// TwinCAT 3 PLC project TwinCAT_OpenFramework_JSON
// Title: TwinCAT Open Framework JSON
// Company: Oleksandr Tiutyk FOP
// Author: Oleksandr Tiutyk
// ProjectVersion: 1.0.13.0
// Description: TwinCAT.OpenFramework сlasses that help in working with JSON
// ProgramVersion: 3.1.4026.28
// libraries:
//   Tc2_Utilities, * (Beckhoff Automation GmbH)
//   Tc3_JsonXml, * (Beckhoff Automation GmbH)
//   [TwinCAT Open Framework Core], * (Oleksandr Tiutyk FOP)
// project tree:
//   AutomaticSerializer/ AutomaticJsonSerializer.TcPOU, IJsonExtender.TcIO
//   Configuration/ JsonConfigurationReader.TcPOU, JsonConfigurationWriter.TcPOU
//   Internal/ CurrentNamespace.TcPOU, JsonDatatypes.TcPOU, NamespaceExtractor.TcPOU
//   Version/ Global_Version.TcGVL
// (motion and I/O tree: see PLC project twincat_openframework_core)
// real-time tasks:
//   TASK PlcTask: cycle T#10ms, priority 20, ADS port 350
//   TASK TestTask: cycle T#10ms, priority 1, ADS port 351
//   TASK RunnerTestTask: cycle T#10ms, priority 2, ADS port 354
//   TASK HowToTask: cycle T#10ms, priority 22, ADS port 353
// variable links:

// ---- Version/Global_Version.TcGVL
{attribute 'TcGenerated'}
{attribute 'no-analysis'}
{attribute 'linkalways'}
// This function has been automatically generated from the project information.
VAR_GLOBAL CONSTANT
	{attribute 'const_non_replaced'}
	stLibVersion_TwinCAT_Open_Framework_JSON : ST_LibVersion := (iMajor := 1, iMinor := 0, iBuild := 13, iRevision := 0, nFlags := 0, sVersion := '1.0.13.0');
END_VAR

// ---- AutomaticSerializer/IJsonExtender.TcIO
(*
SPDX-FileCopyrightText: © 2026 Oleksandr Tiutyk <trofimich@gmail.com>
SPDX-License-Identifier: MIT
License: https://opensource.org/license/mit
*)

(*!
<summary>Extends serialization by writing around the structure's JSON value.</summary>
<description>
AutomaticJsonSerializer calls these hooks synchronously on its own SAX writer. The writer belongs to the
serializer; callbacks do not acquire ownership. The combined hook output and structure value must form the
intended JSON document. The writer is borrowed only for the duration of each callback and must not be retained
or handed to another task. Hooks execute in the serializer's owner task. Do not call methods or access
properties of the active serializer, directly or indirectly; a nested conversion needs a separate serializer
and separate buffers. Stateful extenders must not be used concurrently by different tasks. Implementations
handle failures reported by the native methods they invoke. Callback exceptions propagate from Create methods
and are contained by TrySerialize methods; prior writes and external callback effects are not rolled back.
WriteSuffix is not a cleanup or finally callback.
</description>
*)
INTERFACE IJsonExtender

(*!
<summary>Writes the prefix before serialization of the structure value.</summary>
<description>
Called after successful ResetDocument, before AddJsonValueFromSymbol. Leave the writer ready to receive the
structure as a JSON value, for example after an enclosing container's key. A later failure does not guarantee a
WriteSuffix call or roll back callback effects.
</description>
<param name="jsonSaxWriter">Serializer-owned writer reset for the current conversion.</param>
*)
METHOD WritePrefix
VAR_IN_OUT CONSTANT
	jsonSaxWriter : Tc3_JsonXml.FB_JsonSaxWriter;	
END_VAR
END_METHOD

(*!
<summary>Writes the suffix after successful serialization of the structure value.</summary>
<description>
Called before copying the document to the caller's buffer. May finish a container opened by WritePrefix. It
is skipped if reset, the start hook or structure serialization fails, including terminal allocation failure
contained inside a hook. Later copy failure does not roll back its effects.
</description>
<param name="jsonSaxWriter">Serializer-owned writer containing the prefix and structure value.</param>
*)
METHOD WriteSuffix
VAR_IN_OUT CONSTANT
	jsonSaxWriter : Tc3_JsonXml.FB_JsonSaxWriter;	
END_VAR
END_METHOD

END_INTERFACE

// ---- AutomaticSerializer/AutomaticJsonSerializer.TcPOU
(*
SPDX-FileCopyrightText: © 2026 Oleksandr Tiutyk <trofimich@gmail.com>
SPDX-License-Identifier: MIT
License: https://opensource.org/license/mit
*)

(*!
<summary>Serializes live PLC structures to JSON and restores them from JSON.</summary>
<description>
Supports live PLC structures with native type information; dynamically created structures are not supported.
ByVarInfo methods require an explicit PVOID address; descriptor ByteAddress is ignored to preserve pointer width.
Application method calls and property access belong to one owner task per instance. Instances are not
thread-safe and do not support reentry: a callback must not call methods or access properties of the
serializer whose operation is still active, directly or indirectly. Use a separate instance and separate
buffers for another task or nested conversion. Ownership is a caller precondition, not a runtime check or
lock; Try does not make an ownership violation safe or guarantee its detection as FALSE. Keep source data
stable and destination storage exclusive for the entire call, including callbacks. Separate serializer
instances do not synchronize shared application data. Stateful extenders require their own ownership
discipline; sharing an extender must not introduce concurrent state access. Borrows input, output and optional
callbacks for each call. Throwing methods report invalid arguments and native failures through framework
exceptions. Try methods return FALSE directly for rejected arguments or reported native failures and contain
exceptions from native calls or callbacks; partial effects are not rolled back. Try methods use the shared
native conversion helpers, not overrides of the throwing methods or their protected helpers. JSON text uses
native UTF-8 encoding; capacity and copy sizes count bytes. Instances must not be copied by value. The caller
provides cyclic-task exception cleanup and RaiseIfAllocationFailed at the task boundary, outside Try and
recoverable handlers. Try methods do not clear terminal allocation state. Ownership examples and future
shared-service guidance: Guides/JsonAndEventLoggerOwnership.md in the repository.
</description>
*)

{attribute 'no_explicit_call' := 'Direct call is not allowed'}
FUNCTION_BLOCK AutomaticJsonSerializer EXTENDS TOF_Core.Object
VAR_STAT
	//! <summary>Class name shared by all instances of this function block.</summary>
	{attribute 'hide'} 
	_ClassName : STRING := __POUNAME();
END_VAR
VAR
	_JsonSaxWriter : Tc3_JsonXml.FB_JsonSaxWriter;
	_JsonDataTypeWriter : Tc3_JsonXml.FB_JsonReadWriteDatatype;
END_VAR

(*!
<summary>Provides the concrete serializer class name.</summary>
<description>Borrows read-only instance storage that remains valid for the instance lifetime.</description>
*)
{attribute 'monitoring' := 'call'}
PROPERTY ClassName : REFERENCE TO STRING
GET
ClassName REF= _ClassName;
END_GET
END_PROPERTY

(*!
<summary>Serializes a PLC structure into caller-owned JSON storage.</summary>
<description>
Uses native symbol lookup for the source type; dynamically created structures are not supported. Single-field
structures have native lookup limitations; use ByVarInfo to supply the type explicitly. Borrows
source, destination and optional extender for the call. The destination must be writable and have at least
JSON_DOCUMENT capacity. Invalid source arguments and reported native failures raise framework exceptions;
extender exceptions propagate. Output and callback effects are not rolled back on failure. Exception transport
and cleanup require the caller's cyclic-task boundary. CopyDocument returning zero or a nonzero HRESULT raises
an exception; jsonSize is not usable on failure.
</description>
<param name="sourceStructure">Live PLC structure with type information available to native symbol lookup.</param>
<param name="extender">
Optional callback invoked before and after writing the structure value; zero skips both calls.
</param>
<param name="targetJson">Writable output storage with at least 25000 bytes of text capacity plus the terminator.</param>
<param name="jsonSize">
Byte count reported by CopyDocument, including the terminator on a successful copy; use only after normal
completion.
</param>
*)
METHOD Serialize
VAR_INPUT
	sourceStructure : ANY;
	extender : IJsonExtender := 0;
END_VAR
VAR_IN_OUT
	targetJson : TOF_Core.JSON_DOCUMENT;
END_VAR
VAR_OUTPUT
	jsonSize : UDINT; 
END_VAR
InternalSerialize(
	sourceStructure := sourceStructure,
	extender := extender,
	targetJson := targetJson,
	jsonSize => jsonSize
);
END_METHOD

(*!
<summary>Serializes a PLC structure described by VAR_INFO into caller-owned JSON storage.</summary>
<description>
The descriptor type and byte-aligned size must match sourceStructureAddress. ByteAddress is ignored.
Dynamically created structures are not supported. Borrows source, destination and optional extender for the call. The
destination must be writable and have at least JSON_DOCUMENT capacity. Invalid source arguments and reported
native failures raise framework exceptions; extender exceptions propagate. Output and callback effects are not
rolled back on failure. Exception transport and cleanup require the caller's cyclic-task boundary.
CopyDocument returning zero or a nonzero HRESULT raises an exception; jsonSize is not usable on failure.
</description>
<param name="sourceStructureAddress">
Required address from ADR of the live source structure, borrowed for this call. Must match the descriptor.
Zero is rejected; no address is recovered from ByteAddress or ByteOffset.
</param>
<param name="sourceStructureVarInfo">
Descriptor whose TypeName and BitSize describe the source structure; ByteAddress is ignored.
</param>
<param name="extender">
Optional callback invoked before and after writing the structure value; zero skips both calls.
</param>
<param name="targetJson">Writable output storage with at least 25000 bytes of text capacity plus the terminator.</param>
<param name="jsonSize">
Byte count reported by CopyDocument, including the terminator on a successful copy; use only after normal
completion.
</param>
*)
METHOD SerializeByVarInfo
VAR_INPUT
	sourceStructureVarInfo : __SYSTEM.VAR_INFO;
	sourceStructureAddress : PVOID;
	extender : IJsonExtender := 0;
END_VAR
VAR_IN_OUT
	targetJson : TOF_Core.JSON_DOCUMENT;
END_VAR
VAR_OUTPUT
	jsonSize : UDINT; 
END_VAR
VAR
	formattedExceptionMessage : TOF_Core.ERROR_MESSAGE;

	
	errorCode : HRESULT;
END_VAR
IF sourceStructureAddress = TOF_Core.Memory.NULL_ADDRESS THEN
	TOF_Core.Exceptions.ThrowArgumentNotSpecified(
		sourceNamespaceName := NamespaceName,
		sourceClassName := ClassName,
		sourcePOUName := __POUNAME(),
		sourcePosition := __POSITION(),
		argumentName := 'sourceStructureAddress'
	);
END_IF

IF sourceStructureVarInfo.TypeClass <> __SYSTEM.TYPE_CLASS.TYPE_USERDEF THEN
	TOF_Core.Exceptions.ThrowArgumentTypeClassNotSupported(
		sourceNamespaceName := NamespaceName,
		sourceClassName := ClassName,
		sourcePOUName := __POUNAME(),
		sourcePosition := __POSITION(),
		argumentName := 'sourceStructureVarInfo',
		argumentType := sourceStructureVarInfo.TypeClass
	);
END_IF

// VAR_INFO sizes are in bits; the caller supplies a byte-aligned structure descriptor.
IF NOT writeStructureJson(
	structureTypeName := sourceStructureVarInfo.TypeName,
	structureAddress := sourceStructureAddress,
	structureSize := TO_UDINT(sourceStructureVarInfo.BitSize / 8),
	extender := extender,
	targetJson := targetJson,
	jsonSize => jsonSize,
	errorCode => errorCode,
	errorMessage => formattedExceptionMessage
)
THEN
	TOF_Core.Exceptions.ThrowStandard(
		sourceNamespaceName := NamespaceName,
		sourceClassName := ClassName,
		sourcePOUName := __POUNAME(),
		sourcePosition := __POSITION(),
		message := formattedExceptionMessage,
		errorCode := TO_UDINT(errorCode)
	);
END_IF
END_METHOD

{attribute 'monitoring' := 'call'}
(*!
<summary>Gets or sets the native writer's maximum number of fractional decimal places.</summary>
<description>
The native writer determines which DINT values it supports; this property does not clamp the value. The setter
requires a zero HRESULT from SetMaxDecimalPlaces. A nonzero HRESULT raises a framework exception because
assignment has no failure result. The native error code is retained in the exception. No rollback of the
native setting is guaranteed on failure; the getter reads the writer's current setting. The caller handles the
exception and provides cyclic-task exception cleanup and the terminal allocation-failure boundary.
</description>
*)
PROPERTY DecimalPlaces : DINT
GET
DecimalPlaces := _JsonSaxWriter.GetMaxDecimalPlaces();
END_GET
SET
VAR
	errorCode : HRESULT;
END_VAR
errorCode := _JsonSaxWriter.SetMaxDecimalPlaces(decimalPlaces := DecimalPlaces);

IF errorCode <> TOF_Core.SignedInt32.ZERO THEN
	TOF_Core.Exceptions.ThrowStandard(
		sourceNamespaceName := NamespaceName,
		sourceClassName := ClassName,
		sourcePOUName := __POUNAME(),
		sourcePosition := __POSITION(),
		message := "Can't set JSON writer decimal places",
		errorCode := TO_UDINT(errorCode)
	);
END_IF
END_SET
END_PROPERTY

(*!
<summary>Populates a PLC structure from JSON using the type supplied by VAR_INFO.</summary>
<description>
TypeName and byte-aligned BitSize must describe the live, writable structure at targetStructureAddress.
ByteAddress is ignored. Uses the supplied TypeName directly, avoiding ambiguous address-based type lookup
for single-field structures. The type
must be available to the native JSON converter; support for dynamically created structures is not implied.
Borrows the JSON and destination for this call. A zero address, an unsupported type class or a reported native
conversion failure raises a framework exception. Conversion requires both a TRUE SetSymbolFromJson result and
a zero HRESULT. Destination fields may already have changed on failure; writes are not rolled back. The caller
provides cyclic-task exception cleanup and the terminal allocation-failure boundary.
</description>
<param name="json">JSON text to read without modification.</param>
<param name="targetStructureAddress">
Required address from ADR of the live target structure, borrowed for this call. Must match the descriptor.
Zero is rejected; no address is recovered from ByteAddress or ByteOffset.
</param>
<param name="targetStructureVarInfo">
Consistent descriptor of the destination structure, including its explicit TypeName.
</param>
*)
METHOD DeserializeByVarInfo
VAR_IN_OUT CONSTANT
	json : TOF_Core.JSON_DOCUMENT;	
END_VAR
VAR_INPUT
	targetStructureVarInfo : __SYSTEM.VAR_INFO;
	targetStructureAddress : PVOID;
END_VAR
VAR
	
	errorCode : HRESULT;
END_VAR
IF targetStructureAddress = TOF_Core.Memory.NULL_ADDRESS THEN
	TOF_Core.Exceptions.ThrowArgumentNotSpecified(
		sourceNamespaceName := NamespaceName,
		sourceClassName := ClassName,
		sourcePOUName := __POUNAME(),
		sourcePosition := __POSITION(),
		argumentName := 'targetStructureAddress'
	);
END_IF

IF targetStructureVarInfo.TypeClass <> __SYSTEM.TYPE_CLASS.TYPE_USERDEF THEN
	TOF_Core.Exceptions.ThrowArgumentTypeClassNotSupported(
		sourceNamespaceName := NamespaceName,
		sourceClassName := ClassName,
		sourcePOUName := __POUNAME(),
		sourcePosition := __POSITION(),
		argumentName := 'targetStructureVarInfo',
		argumentType := targetStructureVarInfo.TypeClass
	);
END_IF

// VAR_INFO sizes are in bits; the caller supplies a byte-aligned structure descriptor.
IF NOT readStructureJson(
	json := json,
	structureTypeName := targetStructureVarInfo.TypeName,
	structureAddress := targetStructureAddress,
	structureSize := TO_UDINT(targetStructureVarInfo.BitSize / 8),
	errorCode => errorCode
)
THEN
	TOF_Core.Exceptions.ThrowStandard(
		sourceNamespaceName := NamespaceName,
		sourceClassName := ClassName,
		sourcePOUName := __POUNAME(),
		sourcePosition := __POSITION(),
		message := "Can't fill target structure by specified json document",
		errorCode := TO_UDINT(errorCode)
	);
END_IF
END_METHOD

(*!
<summary>Populates a PLC structure from JSON using native address-based type lookup.</summary>
<description>
Borrows the JSON and a live, writable structure for the call; dynamically created structures are not
supported. Native type lookup has limitations for single-field structures. Invalid arguments, reported lookup
failures, a FALSE SetSymbolFromJson result or a nonzero conversion HRESULT raise framework exceptions.
Destination fields may already have changed on failure; writes are not rolled back. The caller provides
cyclic-task exception cleanup and the terminal allocation-failure boundary.
</description>
<param name="json">JSON text to read without modification.</param>
<param name="targetStructure">
Live destination structure with type information available to native symbol lookup.
</param>
*)
METHOD Deserialize
VAR_IN_OUT CONSTANT
	json : TOF_Core.JSON_DOCUMENT;	
END_VAR
VAR_INPUT
	targetStructure : ANY;
END_VAR
InternalDeserialize(json := json, targetStructure := targetStructure);
END_METHOD

(*!
<summary>Serializes a structure using its ANY descriptor and native symbol lookup.</summary>
<description>
The descriptor must identify a live structure with matching address and size; dynamically created structures
are not supported. Native address lookup has limitations for single-field structures. Borrows source,
destination and optional extender for the call. The destination must be writable and have at least
JSON_DOCUMENT capacity. Invalid source arguments and reported native failures raise framework exceptions;
extender exceptions propagate. Output and callback effects are not rolled back on failure. Overrides must
preserve destination capacity and borrowing requirements. This protected hook serves the throwing ANY API;
TrySerialize does not dispatch through it. Exception transport and cleanup require the caller's
cyclic-task boundary. CopyDocument returning zero or a nonzero HRESULT raises an exception; jsonSize is not
usable on failure.
</description>
<param name="sourceStructure">ANY descriptor for the source structure.</param>
<param name="extender">
Optional callback invoked before and after writing the structure value; zero skips both calls.
</param>
<param name="targetJson">Writable output storage with at least 25000 bytes of text capacity plus the terminator.</param>
<param name="jsonSize">
Byte count reported by CopyDocument, including the terminator on a successful copy; use only after normal
completion.
</param>
*)
METHOD PROTECTED InternalSerialize
VAR_INPUT
	sourceStructure : __SYSTEM.AnyType;
	extender : IJsonExtender := 0;
END_VAR
VAR_IN_OUT
	targetJson : TOF_Core.JSON_DOCUMENT;
END_VAR
VAR_OUTPUT
	jsonSize : UDINT; 
END_VAR
VAR
	formattedExceptionMessage : TOF_Core.ERROR_MESSAGE;

	
	structureTypeName : STRING;	 
	errorCode : HRESULT;
END_VAR
IF sourceStructure.pValue = TOF_Core.Memory.NULL_ADDRESS THEN
	TOF_Core.Exceptions.ThrowArgumentNotSpecified(
		sourceNamespaceName := NamespaceName,
		sourceClassName := ClassName,
		sourcePOUName := __POUNAME(),
		sourcePosition := __POSITION(),
		argumentName := 'sourceStructure'
	);
END_IF

IF sourceStructure.TypeClass <> __SYSTEM.TYPE_CLASS.TYPE_USERDEF THEN
	TOF_Core.Exceptions.ThrowArgumentTypeClassNotSupported(
		sourceNamespaceName := NamespaceName,
		sourceClassName := ClassName,
		sourcePOUName := __POUNAME(),
		sourcePosition := __POSITION(),
		argumentName := 'sourceStructure',
		argumentType := sourceStructure.TypeClass
	);
END_IF

structureTypeName := _JsonDataTypeWriter.GetDatatypeNameByAddress(
	nData := TO_UDINT(sourceStructure.diSize),
	pData := sourceStructure.pValue,
	hrErrorCode => errorCode
);

IF errorCode <> TOF_Core.SignedInt32.ZERO THEN
	TOF_Core.Exceptions.ThrowStandard(
		sourceNamespaceName := NamespaceName,
		sourceClassName := ClassName,
		sourcePOUName := __POUNAME(),
		sourcePosition := __POSITION(),
		message := "Can't get structure type of the source structure",
		errorCode := TO_UDINT(errorCode)
	);
END_IF

IF NOT writeStructureJson(
	structureTypeName := structureTypeName,
	structureAddress := sourceStructure.pValue,
	structureSize := TO_UDINT(sourceStructure.diSize),
	extender := extender,
	targetJson := targetJson,
	jsonSize => jsonSize,
	errorCode => errorCode,
	errorMessage => formattedExceptionMessage
)
THEN
	TOF_Core.Exceptions.ThrowStandard(
		sourceNamespaceName := NamespaceName,
		sourceClassName := ClassName,
		sourcePOUName := __POUNAME(),
		sourcePosition := __POSITION(),
		message := formattedExceptionMessage,
		errorCode := TO_UDINT(errorCode)
	);
END_IF
END_METHOD

(*!
<summary>Deserializes JSON into the structure identified by an ANY descriptor.</summary>
<description>
The descriptor must identify a live, writable structure with matching address and size; dynamically created
structures are not supported. Native address-based type lookup has limitations for single-field structures.
Borrows the JSON and destination for the call. Invalid arguments, reported lookup failures, a FALSE
SetSymbolFromJson result or a nonzero conversion HRESULT raise framework exceptions. Partial destination
writes are not rolled back. Overrides must preserve borrowing and failure reporting requirements. This
protected hook serves the throwing ANY API; TryDeserialize does not dispatch through it. The caller
provides cyclic-task exception cleanup and the terminal allocation-failure boundary.
</description>
<param name="json">JSON text to read without modification.</param>
<param name="targetStructure">ANY descriptor for the live destination structure.</param>
*)
METHOD PROTECTED InternalDeserialize
VAR_IN_OUT CONSTANT
	json : TOF_Core.JSON_DOCUMENT;	
END_VAR
VAR_INPUT
	targetStructure : __SYSTEM.AnyType;
END_VAR
VAR
	
	structureTypeName : STRING;	 
	errorCode : HRESULT;
END_VAR
IF targetStructure.pValue = TOF_Core.Memory.NULL_ADDRESS THEN
	TOF_Core.Exceptions.ThrowArgumentNotSpecified(
		sourceNamespaceName := NamespaceName,
		sourceClassName := ClassName,
		sourcePOUName := __POUNAME(),
		sourcePosition := __POSITION(),
		argumentName := 'targetStructure'
	);
END_IF

IF targetStructure.TypeClass <> __SYSTEM.TYPE_CLASS.TYPE_USERDEF THEN
	TOF_Core.Exceptions.ThrowArgumentTypeClassNotSupported(
		sourceNamespaceName := NamespaceName,
		sourceClassName := ClassName,
		sourcePOUName := __POUNAME(),
		sourcePosition := __POSITION(),
		argumentName := 'targetStructure',
		argumentType := targetStructure.TypeClass
	);
END_IF

structureTypeName := _JsonDataTypeWriter.GetDatatypeNameByAddress(
	nData := TO_UDINT(targetStructure.diSize),
	pData := targetStructure.pValue,
	hrErrorCode => errorCode
);

IF errorCode <> TOF_Core.SignedInt32.ZERO THEN
	TOF_Core.Exceptions.ThrowStandard(
		sourceNamespaceName := NamespaceName,
		sourceClassName := ClassName,
		sourcePOUName := __POUNAME(),
		sourcePosition := __POSITION(),
		message := "Can't get structure type of the target structure",
		errorCode := TO_UDINT(errorCode)
	);
END_IF

IF NOT readStructureJson(
	json := json,
	structureTypeName := structureTypeName,
	structureAddress := targetStructure.pValue,
	structureSize := TO_UDINT(targetStructure.diSize),
	errorCode => errorCode
)
THEN
	TOF_Core.Exceptions.ThrowStandard(
		sourceNamespaceName := NamespaceName,
		sourceClassName := ClassName,
		sourcePOUName := __POUNAME(),
		sourcePosition := __POSITION(),
		message := "Can't fill target structure by specified json document",
		errorCode := TO_UDINT(errorCode)
	);
END_IF
END_METHOD

(*!
<summary>Provides the compiler-initialized library namespace.</summary>
<description>Borrows read-only library storage; no allocation or ownership transfer occurs.</description>
*)
{attribute 'monitoring' := 'call'}
PROPERTY NamespaceName : REFERENCE TO STRING
GET
NamespaceName REF= CurrentNamespace.Name;
END_GET
END_PROPERTY

(*!
<summary>Reads JSON into a validated structure and reports the native conversion result.</summary>
<description>
Callers validate the descriptor before entry. Borrows the JSON, type name and destination for this call.
Returns FALSE for a native FALSE result or nonzero HRESULT without creating exceptions. Native exceptions
propagate to the throwing caller or the public Try boundary. Checks fatal allocation state before conversion
and before reporting success, raising a contained terminal failure without constructing an exception object.
The Try boundary converts that failure to FALSE. Partial destination writes are not rolled back.
</description>
<param name="json">JSON text to read without modification.</param>
<param name="structureTypeName">Native type name matching the destination structure.</param>
<param name="structureAddress">Address of the validated writable destination.</param>
<param name="structureSize">Destination structure size in bytes.</param>
<param name="errorCode">Native conversion HRESULT, interpreted together with the BOOL result.</param>
*)
METHOD PRIVATE readStructureJson : BOOL
VAR_IN_OUT CONSTANT
	json : TOF_Core.JSON_DOCUMENT;
	structureTypeName : STRING;
END_VAR
VAR_INPUT
	structureAddress : PVOID;
	structureSize : UDINT;
END_VAR
VAR_OUTPUT
	errorCode : HRESULT;
END_VAR
TOF_Core.DynamicMemoryManager.RaiseIfAllocationFailed();

IF NOT _JsonDataTypeWriter.SetSymbolFromJson(
		sJson := json,
		sDatatype := structureTypeName,
		nData := structureSize,
		pData := structureAddress,
		hrErrorCode => errorCode
	)
	OR_ELSE errorCode <> TOF_Core.SignedInt32.ZERO
THEN
	RETURN;
END_IF

TOF_Core.DynamicMemoryManager.RaiseIfAllocationFailed();
readStructureJson := TRUE;
END_METHOD

(*!
<summary>Reports the complete instance size in bytes.</summary>
<description>Uses XSIZEOF; separately allocated native resources are not included.</description>
*)
{attribute 'monitoring' := 'call'}
PROPERTY SelfSize : ULINT
GET
SelfSize := XSIZEOF(THIS^);
END_GET
END_PROPERTY

{attribute 'TcRpcEnable':='1'}
(*!
<summary>Attempts to serialize a PLC structure to JSON.</summary>
<description>
Returns FALSE directly for a null address, an unsupported type class or a reported native failure, including a
zero CopyDocument result, without creating a framework exception. Contains native and callback exceptions.
Uses the shared conversion helper rather than the protected throwing hook. Use JSON and jsonSize only on TRUE;
partial writes and callback effects are not rolled back. Each subsequent conversion attempts to reset the
writer before callbacks. Borrows live source and writable destination storage. Does not clear terminal allocation state; the
caller provides exception cleanup and RaiseIfAllocationFailed at the task boundary outside Try and recoverable
handlers. Returns FALSE when fatal allocation state is observed on entry or after nested calls; a contained
allocation failure is not a successful conversion. The application-wide latch remains set.
</description>
<param name="sourceStructure">
Live PLC structure supported by native symbol lookup; dynamically created structures are not supported.
Single-field structures have native lookup limitations; use ByVarInfo to supply the type explicitly.
</param>
<param name="extender">
Optional callback invoked before and after writing the structure value; borrowed for the call.
</param>
<param name="targetJson">
Writable output storage with at least 25000 bytes of text capacity plus the terminator; borrowed for the call.
</param>
<param name="jsonSize">
Byte count reported by CopyDocument, including the terminator on a successful copy; use only on TRUE.
</param>
*)
METHOD TrySerialize : BOOL
VAR_INPUT
	sourceStructure : ANY;
	extender : IJsonExtender := 0;
END_VAR
VAR_IN_OUT
	targetJson : TOF_Core.JSON_DOCUMENT;
END_VAR
VAR_OUTPUT
	jsonSize : UDINT; 
END_VAR
VAR
	structureTypeName : STRING;
	errorCode : HRESULT;
END_VAR
__TRY

	IF TOF_Core.DynamicMemoryManager.HasAllocationFailed THEN
		RETURN;
	END_IF

	IF sourceStructure.pValue = TOF_Core.Memory.NULL_ADDRESS
		OR_ELSE sourceStructure.TypeClass <> __SYSTEM.TYPE_CLASS.TYPE_USERDEF
	THEN
		RETURN;
	END_IF

	structureTypeName := _JsonDataTypeWriter.GetDatatypeNameByAddress(
		nData := TO_UDINT(sourceStructure.diSize),
		pData := sourceStructure.pValue,
		hrErrorCode => errorCode
	);

	IF errorCode <> TOF_Core.SignedInt32.ZERO THEN
		RETURN;
	END_IF

	TrySerialize := writeStructureJson(
		structureTypeName := structureTypeName,
		structureAddress := sourceStructure.pValue,
		structureSize := TO_UDINT(sourceStructure.diSize),
		extender := extender,
		targetJson := targetJson,
		jsonSize => jsonSize
	);

	IF TOF_Core.DynamicMemoryManager.HasAllocationFailed THEN
		TrySerialize := FALSE;
	END_IF

__CATCH
	TrySerialize := FALSE;
__ENDTRY
END_METHOD

(*!
<summary>Attempts to serialize a PLC structure to JSON.</summary>
<description>
Returns FALSE directly for a null address, an unsupported type class or a reported native failure, including a
zero CopyDocument result, without creating a framework exception. Contains native and callback exceptions.
Uses the shared conversion helper rather than the throwing ByVarInfo method. Use JSON and jsonSize only on
TRUE; partial writes and callback effects are not rolled back. Each subsequent conversion attempts to reset
the writer before callbacks. Borrows live source and writable destination storage. Does not clear terminal allocation
state; the caller provides exception cleanup and RaiseIfAllocationFailed at the task boundary outside Try and
recoverable handlers. Returns FALSE when fatal allocation state is observed on entry or after nested calls; a contained
allocation failure is not a successful conversion. The application-wide latch remains set.
</description>
<param name="sourceStructureAddress">
Required address from ADR of the live source structure, borrowed for this call. Must match the descriptor.
Zero is rejected; no address is recovered from ByteAddress or ByteOffset.
</param>
<param name="sourceStructureVarInfo">
Descriptor with matching TypeName and byte-aligned BitSize for sourceStructureAddress; ByteAddress is ignored.
Dynamically created structures are not supported.
</param>
<param name="extender">
Optional callback invoked before and after writing the structure value; borrowed for the call.
</param>
<param name="targetJson">
Writable output storage with at least 25000 bytes of text capacity plus the terminator; borrowed for the call.
</param>
<param name="jsonSize">
Byte count reported by CopyDocument, including the terminator on a successful copy; use only on TRUE.
</param>
*)
METHOD TrySerializeByVarInfo : BOOL
VAR_INPUT
	sourceStructureVarInfo : __SYSTEM.VAR_INFO;
	sourceStructureAddress : PVOID;
	extender : IJsonExtender := 0;
END_VAR
VAR_IN_OUT
	targetJson : TOF_Core.JSON_DOCUMENT;
END_VAR
VAR_OUTPUT
	jsonSize : UDINT; 
END_VAR
__TRY

	IF TOF_Core.DynamicMemoryManager.HasAllocationFailed THEN
		RETURN;
	END_IF

	IF sourceStructureAddress = TOF_Core.Memory.NULL_ADDRESS
		OR_ELSE sourceStructureVarInfo.TypeClass <> __SYSTEM.TYPE_CLASS.TYPE_USERDEF
	THEN
		RETURN;
	END_IF

	// VAR_INFO sizes are in bits; the descriptor must be byte-aligned.
	TrySerializeByVarInfo := writeStructureJson(
		structureTypeName := sourceStructureVarInfo.TypeName,
		structureAddress := sourceStructureAddress,
		structureSize := TO_UDINT(sourceStructureVarInfo.BitSize / 8),
		extender := extender,
		targetJson := targetJson,
		jsonSize => jsonSize
	);

	IF TOF_Core.DynamicMemoryManager.HasAllocationFailed THEN
		TrySerializeByVarInfo := FALSE;
	END_IF

__CATCH
	TrySerializeByVarInfo := FALSE;
__ENDTRY
END_METHOD

(*!
<summary>Attempts to populate a PLC structure from JSON using the type supplied by VAR_INFO.</summary>
<description>
Uses the supplied TypeName directly without address-based type lookup. TypeName and byte-aligned BitSize must
describe the live, writable structure at targetStructureAddress, with its type available to the native converter.
ByteAddress is ignored.
Returns FALSE directly for a null address, an unsupported type class, a FALSE native conversion result or a
nonzero HRESULT, without creating a framework exception. Contains native exceptions. Uses the shared
conversion helper rather than the throwing ByVarInfo method. Partial destination writes are not rolled back.
Borrows the JSON and destination for this call. Does not clear terminal allocation state; the caller provides
exception cleanup and RaiseIfAllocationFailed at the task boundary outside Try and recoverable handlers.
Returns FALSE when fatal allocation state is observed on entry or after nested calls; a contained
allocation failure is not a successful conversion. The application-wide latch remains set.
</description>
<param name="json">JSON text to read without modification.</param>
<param name="targetStructureAddress">
Required address from ADR of the live target structure, borrowed for this call. Must match the descriptor.
Zero is rejected; no address is recovered from ByteAddress or ByteOffset.
</param>
<param name="targetStructureVarInfo">
Consistent descriptor of the destination structure, including its explicit TypeName.
</param>
*)
METHOD TryDeserializeByVarInfo : BOOL
VAR_IN_OUT CONSTANT
	json : TOF_Core.JSON_DOCUMENT;	
END_VAR
VAR_INPUT
	targetStructureVarInfo : __SYSTEM.VAR_INFO;
	targetStructureAddress : PVOID;
END_VAR
__TRY

	IF TOF_Core.DynamicMemoryManager.HasAllocationFailed THEN
		RETURN;
	END_IF

	IF targetStructureAddress = TOF_Core.Memory.NULL_ADDRESS
		OR_ELSE targetStructureVarInfo.TypeClass <> __SYSTEM.TYPE_CLASS.TYPE_USERDEF
	THEN
		RETURN;
	END_IF

	// VAR_INFO sizes are in bits; the descriptor must be byte-aligned.
	TryDeserializeByVarInfo := readStructureJson(
		json := json,
		structureTypeName := targetStructureVarInfo.TypeName,
		structureAddress := targetStructureAddress,
		structureSize := TO_UDINT(targetStructureVarInfo.BitSize / 8)
	);

	IF TOF_Core.DynamicMemoryManager.HasAllocationFailed THEN
		TryDeserializeByVarInfo := FALSE;
	END_IF

__CATCH
	TryDeserializeByVarInfo := FALSE;
__ENDTRY
END_METHOD

(*!
<summary>Attempts to populate a PLC structure from JSON.</summary>
<description>
Uses native address-based type lookup, with its limitations for single-field structures; dynamically created
structures are not supported. Returns FALSE directly for a null address, an unsupported type class, a reported
lookup failure, a FALSE native conversion result or a nonzero conversion HRESULT, without creating a framework
exception. Contains native exceptions. Uses the shared conversion helper rather than the protected throwing
hook. Partial destination writes are not rolled back. Borrows JSON and live, writable destination storage for
this call. Does not clear terminal allocation state; the caller provides exception cleanup and
RaiseIfAllocationFailed at the task boundary outside Try and recoverable handlers.
Returns FALSE when fatal allocation state is observed on entry or after nested calls; a contained
allocation failure is not a successful conversion. The application-wide latch remains set.
</description>
<param name="json">JSON text to read without modification.</param>
<param name="targetStructure">
Live destination structure with type information available to native symbol lookup.
</param>
*)
METHOD TryDeserialize : BOOL
VAR_IN_OUT CONSTANT
	json : TOF_Core.JSON_DOCUMENT;	
END_VAR
VAR_INPUT
	targetStructure : ANY;
END_VAR
VAR
	structureTypeName : STRING;
	errorCode : HRESULT;
END_VAR
__TRY

	IF TOF_Core.DynamicMemoryManager.HasAllocationFailed THEN
		RETURN;
	END_IF

	IF targetStructure.pValue = TOF_Core.Memory.NULL_ADDRESS
		OR_ELSE targetStructure.TypeClass <> __SYSTEM.TYPE_CLASS.TYPE_USERDEF
	THEN
		RETURN;
	END_IF

	structureTypeName := _JsonDataTypeWriter.GetDatatypeNameByAddress(
		nData := TO_UDINT(targetStructure.diSize),
		pData := targetStructure.pValue,
		hrErrorCode => errorCode
	);

	IF errorCode <> TOF_Core.SignedInt32.ZERO THEN
		RETURN;
	END_IF

	TryDeserialize := readStructureJson(
		json := json,
		structureTypeName := structureTypeName,
		structureAddress := targetStructure.pValue,
		structureSize := TO_UDINT(targetStructure.diSize)
	);

	IF TOF_Core.DynamicMemoryManager.HasAllocationFailed THEN
		TryDeserialize := FALSE;
	END_IF

__CATCH
	TryDeserialize := FALSE;
__ENDTRY
END_METHOD

(*!
<summary>Writes a validated structure and optional extensions to caller-owned JSON storage.</summary>
<description>
Callers validate the structure descriptor before entry. Borrows all arguments for this call and resets the
writer before invoking callbacks. A nonzero ResetDocument HRESULT returns FALSE before any hook or copy.
Returns FALSE for reported native failures without creating exceptions; native or callback exceptions propagate
to the throwing caller or the public Try boundary. Checks fatal allocation state before native work, after
successful native steps and after each hook. A contained terminal failure is raised again without allocating
an exception object; the Try boundary converts it to FALSE. No output, writer or callback effects are rolled
back. Each later write attempts to reset the writer again. On FALSE, errorMessage describes the failed native
step and errorCode retains its HRESULT without substitution.
</description>
<param name="structureTypeName">Native type name matching the live source structure.</param>
<param name="structureAddress">Address of the validated source structure.</param>
<param name="structureSize">Source structure size in bytes.</param>
<param name="extender">Optional callbacks around the structure value.</param>
<param name="targetJson">Writable storage with JSON_DOCUMENT capacity, including its terminator.</param>
<param name="jsonSize">Copied byte count including the terminator; meaningful only on TRUE.</param>
<param name="errorCode">Native HRESULT of the failed step on FALSE.</param>
<param name="errorMessage">Diagnostic for the failed step on FALSE.</param>
*)
METHOD PRIVATE writeStructureJson : BOOL
VAR_IN_OUT CONSTANT
	structureTypeName : STRING;
END_VAR
VAR_INPUT
	structureAddress : PVOID;
	structureSize : UDINT;
	extender : IJsonExtender;
END_VAR
VAR_IN_OUT
	targetJson : TOF_Core.JSON_DOCUMENT;
END_VAR
VAR_OUTPUT
	jsonSize : UDINT;
	errorCode : HRESULT;
	errorMessage : WSTRING(255);
END_VAR
TOF_Core.DynamicMemoryManager.RaiseIfAllocationFailed();
errorCode := _JsonSaxWriter.ResetDocument();
TOF_Core.DynamicMemoryManager.RaiseIfAllocationFailed();

IF errorCode <> TOF_Core.SignedInt32.ZERO THEN
	errorMessage := "Can't reset JSON writer before structure serialization";
	RETURN;
END_IF

IF extender <> 0 THEN
	extender.WritePrefix(jsonSaxWriter := _JsonSaxWriter);
	TOF_Core.DynamicMemoryManager.RaiseIfAllocationFailed();
END_IF

IF NOT _JsonDataTypeWriter.AddJsonValueFromSymbol(
		fbWriter := _JsonSaxWriter,
		sDatatype := structureTypeName,
		nData := structureSize,
		pData := structureAddress,
		hrErrorCode => errorCode
	)
	OR_ELSE errorCode <> TOF_Core.SignedInt32.ZERO
THEN
	errorMessage := TOF_Core.WideStrings.Concat255(
		"Can't generate JSON representation from the symbol of type '",
		TO_WSTRING(structureTypeName),
		"'"
	);
	RETURN;
END_IF

TOF_Core.DynamicMemoryManager.RaiseIfAllocationFailed();

IF extender <> 0 THEN
	extender.WriteSuffix(jsonSaxWriter := _JsonSaxWriter);
	TOF_Core.DynamicMemoryManager.RaiseIfAllocationFailed();
END_IF

jsonSize := _JsonSaxWriter.CopyDocument(
	pDoc := targetJson,
	nDoc := SIZEOF(targetJson),
	hrErrorCode => errorCode
);

IF jsonSize = TOF_Core.UnsignedInt32.MIN_VALUE OR_ELSE errorCode <> TOF_Core.SignedInt32.ZERO THEN
	errorMessage := TOF_Core.WideStrings.Concat255(
		"Can't fill JSON from the symbol of type '",
		TO_WSTRING(structureTypeName),
		"'"
	);
	RETURN;
END_IF

TOF_Core.DynamicMemoryManager.RaiseIfAllocationFailed();
writeStructureJson := TRUE;
END_METHOD

END_FUNCTION_BLOCK

// ---- Internal/CurrentNamespace.TcPOU
(*
SPDX-FileCopyrightText: © 2026 Oleksandr Tiutyk <trofimich@gmail.com>
SPDX-License-Identifier: MIT
License: https://opensource.org/license/mit
*)

(*!
<summary>Provides this library's namespace text to object metadata getters.</summary>
<description>
Owns the namespace extractor for the program instance's lifetime; no cyclic execution is required.
</description>
*)

{attribute 'no_explicit_call' := 'do not call this POU directly'}
PROGRAM INTERNAL CurrentNamespace
VAR
	{attribute 'hide'} 
	_NamespaceExtractor : NamespaceExtractor;
END_VAR

{attribute 'monitoring' := 'call'}
(*!
<summary>Returns a borrowed reference to the stored namespace text.</summary>
<description>
The reference belongs to this program instance and remains valid while it exists. Callers must treat the text
as read-only; reading does not copy or allocate storage.
</description>
*)
PROPERTY Name : REFERENCE TO STRING
GET
Name REF= _NamespaceExtractor.CurrentNamespace;
END_GET
END_PROPERTY

END_PROGRAM

// ---- Internal/NamespaceExtractor.TcPOU
(*
SPDX-FileCopyrightText: © 2026 Oleksandr Tiutyk <trofimich@gmail.com>
SPDX-License-Identifier: MIT
License: https://opensource.org/license/mit
*)

(*!
<summary>Holds namespace text initialized through the init_namespace attribute.</summary>
<description>
The compiler supplies the initial text; this block performs no runtime extraction or allocation. The owning
CurrentNamespace program exposes the stored text as borrowed metadata.
</description>
*)

FUNCTION_BLOCK INTERNAL NamespaceExtractor
VAR_OUTPUT
	//! <summary>Compiler-initialized namespace storage; consumers must not modify it.</summary>
	{attribute 'init_namespace'} 
	CurrentNamespace : STRING; 	
END_VAR

END_FUNCTION_BLOCK

// ---- Configuration/JsonConfigurationReader.TcPOU
(*
SPDX-FileCopyrightText: © 2026 Oleksandr Tiutyk <trofimich@gmail.com>
SPDX-License-Identifier: MIT
License: https://opensource.org/license/mit
*)

(*!
<summary>Reads a JSON document using scoped DOM handles.</summary>
<description>
Use a single instance from one task without reentry. UTF-8 text, including ASCII and empty strings, is decoded directly.
Legacy encodings use the native symbol converter.
</description>
*)

{attribute 'no_explicit_call' := 'do not call this function block directly'}
FUNCTION_BLOCK JsonConfigurationReader EXTENDS TOF_Core.Object IMPLEMENTS TOF_Core.IConfigurationReader
VAR_STAT
	_ClassName : STRING := __POUNAME();
END_VAR
VAR
	_Parser : Tc3_JsonXml.FB_JsonDomParser;
	_Converter : Tc3_JsonXml.FB_JsonReadWriteDatatype;
	_Value : TOF_Core.JSON_DOCUMENT;
END_VAR

(*!
<summary>Provides the concrete serializer class name.</summary>
<description>Borrows read-only instance storage that remains valid for the instance lifetime.</description>
*)
{attribute 'monitoring' := 'call'}
PROPERTY ClassName : REFERENCE TO STRING
GET
ClassName REF= _ClassName;
END_GET
END_PROPERTY

(*!
<summary>Attempts to find an optional object member without throwing.</summary>
<description>Returns EMPTY_NODE when absent. No exception escapes this method.</description>
<param name="node">Parent object node.</param>
<param name="name">Optional member field name.</param>
*)
METHOD FindField : TOF_Core.CONFIGURATION_NODE
VAR_INPUT
	node : TOF_Core.CONFIGURATION_NODE;
	name : STRING;
END_VAR
VAR
	member : __XWORD;
END_VAR
IF node.Handle = 0 OR_ELSE NOT _Parser.IsObject(v := node.Handle) THEN
	FindField := TOF_Core.ConfigurationNodes.EMPTY_NODE;
	RETURN;
END_IF

member := _Parser.FindMember(v := node.Handle, member := name);
FindField.Handle := member;
END_METHOD

(*!
<summary>Returns the number of elements of an array. Other shapes raise.</summary>
<description>
Use within one synchronous load. Handles borrow the active document and expire when it is replaced.
</description>
<param name="node">Array node.</param>
*)
METHOD GetArraySize : UDINT
VAR_INPUT
	node : TOF_Core.CONFIGURATION_NODE;
END_VAR
IF NOT IsArray(node := node) THEN
	throwInvalidDocumentException(reason := 'not an array', fieldName := '');
END_IF

GetArraySize := _Parser.GetArraySize(v := node.Handle);
END_METHOD

(*!
<summary>Finds a mandatory object member or raises.</summary>
<description>
Use within one synchronous load. Handles borrow the active document and expire when it is replaced.
</description>
<param name="node">Parent object node.</param>
<param name="name">Member field name.</param>
*)
METHOD GetField : TOF_Core.CONFIGURATION_NODE
VAR_INPUT
	node : TOF_Core.CONFIGURATION_NODE;
	name : STRING;
END_VAR
IF node.Handle = 0 OR_ELSE NOT _Parser.IsObject(v := node.Handle) THEN
	throwInvalidDocumentException(reason := 'not an object', fieldName := name);
END_IF

GetField.Handle := _Parser.FindMember(v := node.Handle, member := name);

IF GetField.Handle = 0 THEN
	throwInvalidDocumentException(reason := 'missing field', fieldName := name);
END_IF
END_METHOD

(*!
<summary>Returns an existing array item by zero-based index or raises.</summary>
<description>Use within one synchronous load. Out-of-bounds index raises an exception.</description>
<param name="node">Array node.</param>
<param name="index">Zero-based element index.</param>
*)
METHOD GetItem : TOF_Core.CONFIGURATION_NODE
VAR_INPUT
	node : TOF_Core.CONFIGURATION_NODE;
	index : UDINT;
END_VAR
IF NOT IsArray(node := node) THEN
	throwInvalidDocumentException(reason := 'not an array', fieldName := '');
END_IF

IF index >= _Parser.GetArraySize(v := node.Handle) THEN
	throwInvalidDocumentException(reason := 'index out of range', fieldName := '');
END_IF

GetItem.Handle := _Parser.GetArrayValueByIdx(v := node.Handle, idx := index);
END_METHOD

(*!
<summary>Reports whether the supplied value is an array.</summary>
<description>
Use within one synchronous load. Handles borrow the active document and expire when it is replaced.
</description>
<param name="node">Node to inspect.</param>
*)
METHOD IsArray : BOOL
VAR_INPUT
	node : TOF_Core.CONFIGURATION_NODE;
END_VAR
IsArray := node.Handle <> 0 AND_THEN _Parser.IsArray(v := node.Handle);
END_METHOD

(*!
<summary>Reports whether the supplied node refers to a present document element.</summary>
<description>Returns FALSE for an empty or unassigned node handle.</description>
<param name="node">Node to inspect.</param>
*)
METHOD IsPresent : BOOL
VAR_INPUT
	node : TOF_Core.CONFIGURATION_NODE;
END_VAR
IsPresent := node.Handle <> 0;
END_METHOD

(*!
<summary>Provides the compiler-initialized library namespace.</summary>
<description>Borrows read-only library storage; no allocation or ownership transfer occurs.</description>
*)
{attribute 'monitoring' := 'call'}
PROPERTY NamespaceName : REFERENCE TO STRING
GET
NamespaceName REF= CurrentNamespace.Name;
END_GET
END_PROPERTY

(*!
<summary>Parses a JSON configuration document and returns its root cursor node.</summary>
<description>Requires an object root. A new call invalidates all previously issued cursors.</description>
<param name="document">Null-terminated JSON document text.</param>
*)
METHOD Parse : TOF_Core.CONFIGURATION_NODE
VAR_IN_OUT CONSTANT
	document : TOF_Core.JSON_DOCUMENT;
END_VAR
Parse.Handle := _Parser.ParseDocument(sJson := document);

IF Parse.Handle = 0 THEN
	throwInvalidDocumentException(reason := 'parse failure', fieldName := '');
ELSIF NOT _Parser.IsObject(v := Parse.Handle) THEN
	throwInvalidDocumentException(reason := 'not an object', fieldName := '');
END_IF
END_METHOD

(*!
<summary>Reads one elementary value into a live typed destination or raises.</summary>
<description>
Use within one synchronous load. Handles borrow the active document and expire when it is replaced.
WSTRING requires a JSON string. Direct UTF-8 decoding checks the destination capacity before writing.
Native copy failures identify the operation and buffer size. Read the destination only after successful return.
</description>
<param name="node">Node containing the elementary value.</param>
<param name="valueType">Elementary IEC type class to decode.</param>
<param name="data">Writable pointer to the destination memory.</param>
<param name="size">Destination memory size in bytes.</param>
*)
METHOD ReadValue
VAR_INPUT
	node : TOF_Core.CONFIGURATION_NODE;
	valueType : TOF_Core.CONFIGURATION_VALUE_TYPE;
	data : PVOID;
	size : UDINT;
END_VAR
VAR
	typeName : STRING;
	target : POINTER TO STRING;
	result : HRESULT;
END_VAR
IF data = 0 OR_ELSE size = 0 THEN
	throwInvalidDocumentException(reason := 'type/size mismatch', fieldName := '');
END_IF

IF node.Handle = 0 THEN
	throwInvalidDocumentException(reason := 'missing field', fieldName := '');
END_IF

IF _Parser.IsNull(v := node.Handle)
	OR_ELSE _Parser.IsArray(v := node.Handle)
	OR_ELSE _Parser.IsObject(v := node.Handle)
THEN
	throwInvalidDocumentException(reason := 'type/size mismatch', fieldName := '');
END_IF

typeName := JsonDatatypes.ToDatatypeName(valueType := valueType, size := size);

IF typeName = '' THEN
	throwInvalidDocumentException(reason := 'type/size mismatch', fieldName := '');
END_IF

IF valueType = TOF_Core.CONFIGURATION_VALUE_TYPE.TYPE_STRING THEN
	target := data;

	IF NOT _Parser.IsString(v := node.Handle) THEN
		throwInvalidDocumentException(reason := 'type/size mismatch', fieldName := '');
	END_IF

	IF _Parser.CopyString(v := node.Handle, pStr := target^, nStr := size) = 0 THEN
		throwInvalidDocumentException(
			reason := TOF_Core.Strings.Concat255(
				'CopyString failed for ', typeName, ' (', TO_STRING(size), ' destination bytes)'
			),
			fieldName := ''
		);
	END_IF

	RETURN;
END_IF

IF valueType = TOF_Core.CONFIGURATION_VALUE_TYPE.TYPE_WSTRING THEN
	IF NOT _Parser.IsString(v := node.Handle) THEN
		throwInvalidDocumentException(reason := 'type/size mismatch', fieldName := '');
	END_IF

	IF readUtf8WideString(node := node, destination := data, size := size) THEN
		RETURN;
	END_IF
END_IF

IF _Parser.CopyJson(v := node.Handle, pDoc := _Value, nDoc := SIZEOF(_Value)) = 0 THEN
	throwInvalidDocumentException(
		reason := TOF_Core.Strings.Concat255(
			'CopyJson failed for ', typeName, ' (', TO_STRING(SIZEOF(_Value)), ' JSON buffer bytes)'
		),
		fieldName := ''
	);
END_IF

IF NOT _Converter.SetSymbolFromJson(
	sJson := _Value,
	sDatatype := typeName,
	nData := size,
	pData := data,
	hrErrorCode => result
) OR_ELSE result <> 0 THEN
	throwInvalidDocumentException(reason := 'parse failure', fieldName := '');
END_IF
END_METHOD

(*!
<summary>Reports the complete instance size in bytes.</summary>
<description>Uses XSIZEOF; separately allocated native resources are not included.</description>
*)
{attribute 'monitoring' := 'call'}
PROPERTY SelfSize : ULINT
GET
SelfSize := XSIZEOF(THIS^);
END_GET
END_PROPERTY

(*!
<summary>Decodes a JSON string directly into a WSTRING destination when its bytes are available as UTF-8.</summary>
<description>
Expects a live string node and a writable WSTRING buffer with a validated byte size. Returns FALSE
without writing when the copied text uses a legacy encoding.
The caller then uses the native symbol converter. Inspects JSON escapes before copying decoded text to an IEC string.
Both DOM and copy sizes include the terminator. Rejects a size mismatch,
an embedded null, insufficient destination capacity, or incomplete conversion. Conversion failure may modify the destination.
</description>
*)
METHOD PRIVATE readUtf8WideString : BOOL
VAR_INPUT
	node : TOF_Core.CONFIGURATION_NODE;
	destination : POINTER TO WSTRING;
	size : UDINT;
END_VAR
VAR
	// A JSON escape for U+0000, which IEC text cannot represent within a value.
	nullEscape : STRING(6) := '\u0000';
	jsonSize : UDINT;
	offset : UDINT;
	escapeIndex : UDINT;
	jsonBytes : POINTER TO BYTE;
	domStringSize : UDINT;
	copiedSize : UDINT;
	characterCount : UDINT;
	decodedCount : UDINT;
END_VAR
jsonSize := _Parser.CopyJson(v := node.Handle, pDoc := _Value, nDoc := SIZEOF(_Value));

IF jsonSize = 0 THEN
	throwInvalidDocumentException(reason := 'parse failure', fieldName := '');
END_IF

jsonBytes := ADR(_Value);
offset := 1; // Skip the opening JSON quote.

WHILE offset + SIZEOF(nullEscape) <= jsonSize DO
	IF jsonBytes[offset] = nullEscape[0] THEN
		escapeIndex := 1;

		WHILE escapeIndex < SIZEOF(nullEscape) - TOF_Core.Strings.CharSize
			AND_THEN jsonBytes[offset + escapeIndex] = nullEscape[escapeIndex]
		DO
			escapeIndex := escapeIndex + 1;
		END_WHILE

		IF escapeIndex = SIZEOF(nullEscape) - TOF_Core.Strings.CharSize THEN
			throwInvalidDocumentException(reason := 'parse failure', fieldName := '');
		END_IF

		// Skip the escaped byte as well, including a second backslash in a literal backslash pair.
		offset := offset + 1;
	END_IF

	offset := offset + 1;
END_WHILE

domStringSize := _Parser.GetStringLength(v := node.Handle);

copiedSize := _Parser.CopyString(v := node.Handle, pStr := _Value, nStr := SIZEOF(_Value));

IF copiedSize = 0
	OR_ELSE copiedSize <> domStringSize
	OR_ELSE TOF_Core.Strings.GetActualSize(value := _Value) <> copiedSize
THEN
	throwInvalidDocumentException(reason := 'parse failure', fieldName := '');
END_IF

IF copiedSize = TOF_Core.Strings.CharSize THEN
	destination^[0] := 0;
	readUtf8WideString := TRUE;
	RETURN;
END_IF

characterCount := Tc2_Utilities.UTF8Len(pUTF8 := ADR(_Value));

IF characterCount = 0 THEN
	RETURN;
END_IF

IF characterCount >= size / TOF_Core.WideStrings.CharSize THEN
	throwInvalidDocumentException(
		reason := TOF_Core.Strings.Concat255(
			'WSTRING needs ', TO_STRING(characterCount), ' characters, capacity ',
			TO_STRING(size / TOF_Core.WideStrings.CharSize - 1)
		),
		fieldName := ''
	);
END_IF

IF NOT Tc2_Utilities.UTF8_TO_WSTRING(
	pDstWSTRING := destination,
	pSrcUTF8 := ADR(_Value),
	nDstSize := size,
	nDstLen => decodedCount
) OR_ELSE decodedCount <> characterCount THEN
	throwInvalidDocumentException(reason := 'parse failure', fieldName := '');
END_IF

readUtf8WideString := TRUE;
END_METHOD

(*!
<summary>Reports an invalid or incompatible configuration value or document structure.</summary>
<description>
Constructs a diagnostic error message with the failure cause and optional member name, and raises StandardException.
The reader remains reusable by opening another document.
</description>
<param name="reason">Specific failure description.</param>
<param name="fieldName">Associated member field name, or empty when not applicable.</param>
*)
METHOD PRIVATE throwInvalidDocumentException
VAR_INPUT
	reason : STRING;
	fieldName : STRING;
END_VAR
VAR
	diagnosticMessage : TOF_Core.ERROR_MESSAGE;
END_VAR
IF fieldName <> '' THEN
	diagnosticMessage := TO_WSTRING(TOF_Core.Strings.Concat255(
		'Invalid JSON configuration: ',
		reason,
		' (field: ',
		fieldName,
		')'
	));
ELSE
	diagnosticMessage := TO_WSTRING(TOF_Core.Strings.Concat255('Invalid JSON configuration: ', reason));
END_IF

TOF_Core.Exceptions.ThrowStandard(
	sourceNamespaceName := NamespaceName,
	sourceClassName := ClassName,
	sourcePOUName := __POUNAME(),
	sourcePosition := __POSITION(),
	message := diagnosticMessage,
	errorCode := 16#80070057
);
END_METHOD

END_FUNCTION_BLOCK

// ---- Internal/JsonDatatypes.TcPOU
(*
SPDX-FileCopyrightText: © 2026 Oleksandr Tiutyk <trofimich@gmail.com>
SPDX-License-Identifier: MIT
License: https://opensource.org/license/mit
*)

(*!
<summary>Maps Core configuration value types and byte sizes to Tc3_JsonXml symbol datatype names.</summary>
<description>
Delegates byte-size validation to TOF_Core.ConfigurationValueTypes.IsValidSize before constructing the native
datatype string for FB_JsonReadWriteDatatype. Uses TwinCAT symbol datatype names for time-of-day and datetime values.
</description>
*)

{attribute 'no_explicit_call' := 'do not call this function block directly'}
PROGRAM INTERNAL JsonDatatypes
VAR
	{attribute 'hide'}
	_ClassName : STRING := __POUNAME();
END_VAR

(*!
<summary>Returns the program class name for diagnostic reporting.</summary>
*)
{attribute 'monitoring' := 'call'}
PROPERTY ClassName : REFERENCE TO STRING
GET
ClassName REF= _ClassName;
END_GET
END_PROPERTY

(*!
<summary>Returns the library namespace name for diagnostic reporting.</summary>
*)
{attribute 'monitoring' := 'call'}
PROPERTY NamespaceName : REFERENCE TO STRING
GET
NamespaceName REF= CurrentNamespace.Name;
END_GET
END_PROPERTY

(*!
<summary>Maps a CONFIGURATION_VALUE_TYPE and buffer byte size to a Tc3_JsonXml symbol datatype name.</summary>
<description>
Validates size via TOF_Core.ConfigurationValueTypes.IsValidSize. Returns an empty string when the type or size
is invalid; no exception is raised. Uses the names emitted in TwinCAT symbol metadata for time-of-day and datetime.
</description>
<param name="valueType">Elementary configuration value type.</param>
<param name="size">Buffer size in bytes.</param>
*)
METHOD ToDatatypeName : STRING
VAR_INPUT
	valueType : TOF_Core.CONFIGURATION_VALUE_TYPE;
	size : UDINT;
END_VAR
VAR
	capacity : UDINT;
END_VAR
IF NOT TOF_Core.ConfigurationValueTypes.IsValidSize(valueType := valueType, size := size) THEN
	RETURN;
END_IF

CASE valueType OF
	TOF_Core.CONFIGURATION_VALUE_TYPE.TYPE_BOOL:
		ToDatatypeName := 'BOOL';

	TOF_Core.CONFIGURATION_VALUE_TYPE.TYPE_BYTE:
		ToDatatypeName := 'BYTE';

	TOF_Core.CONFIGURATION_VALUE_TYPE.TYPE_WORD:
		ToDatatypeName := 'WORD';

	TOF_Core.CONFIGURATION_VALUE_TYPE.TYPE_DWORD:
		ToDatatypeName := 'DWORD';

	TOF_Core.CONFIGURATION_VALUE_TYPE.TYPE_LWORD:
		ToDatatypeName := 'LWORD';

	TOF_Core.CONFIGURATION_VALUE_TYPE.TYPE_SINT:
		ToDatatypeName := 'SINT';

	TOF_Core.CONFIGURATION_VALUE_TYPE.TYPE_INT:
		ToDatatypeName := 'INT';

	TOF_Core.CONFIGURATION_VALUE_TYPE.TYPE_DINT:
		ToDatatypeName := 'DINT';

	TOF_Core.CONFIGURATION_VALUE_TYPE.TYPE_LINT:
		ToDatatypeName := 'LINT';

	TOF_Core.CONFIGURATION_VALUE_TYPE.TYPE_USINT:
		ToDatatypeName := 'USINT';

	TOF_Core.CONFIGURATION_VALUE_TYPE.TYPE_UINT:
		ToDatatypeName := 'UINT';

	TOF_Core.CONFIGURATION_VALUE_TYPE.TYPE_UDINT:
		ToDatatypeName := 'UDINT';

	TOF_Core.CONFIGURATION_VALUE_TYPE.TYPE_ULINT:
		ToDatatypeName := 'ULINT';

	TOF_Core.CONFIGURATION_VALUE_TYPE.TYPE_REAL:
		ToDatatypeName := 'REAL';

	TOF_Core.CONFIGURATION_VALUE_TYPE.TYPE_LREAL:
		ToDatatypeName := 'LREAL';

	TOF_Core.CONFIGURATION_VALUE_TYPE.TYPE_TIME:
		ToDatatypeName := 'TIME';

	TOF_Core.CONFIGURATION_VALUE_TYPE.TYPE_LTIME:
		ToDatatypeName := 'LTIME';

	TOF_Core.CONFIGURATION_VALUE_TYPE.TYPE_DATE:
		ToDatatypeName := 'DATE';

	TOF_Core.CONFIGURATION_VALUE_TYPE.TYPE_LDATE:
		ToDatatypeName := 'LDATE';

	TOF_Core.CONFIGURATION_VALUE_TYPE.TYPE_TOD:
		ToDatatypeName := 'TIME_OF_DAY';

	TOF_Core.CONFIGURATION_VALUE_TYPE.TYPE_LTOD:
		ToDatatypeName := 'LTIME_OF_DAY';

	TOF_Core.CONFIGURATION_VALUE_TYPE.TYPE_DT:
		ToDatatypeName := 'DATE_AND_TIME';

	TOF_Core.CONFIGURATION_VALUE_TYPE.TYPE_LDT:
		ToDatatypeName := 'LDATE_AND_TIME';

	TOF_Core.CONFIGURATION_VALUE_TYPE.TYPE_STRING:
		capacity := size - 1;
		ToDatatypeName := TOF_Core.Strings.Concat255('STRING(', TO_STRING(capacity), ')');

	TOF_Core.CONFIGURATION_VALUE_TYPE.TYPE_WSTRING:
		capacity := (size / 2) - 1;
		ToDatatypeName := TOF_Core.Strings.Concat255('WSTRING(', TO_STRING(capacity), ')');
END_CASE
END_METHOD

END_PROGRAM

// ---- Configuration/JsonConfigurationWriter.TcPOU
(*
SPDX-FileCopyrightText: © 2026 Oleksandr Tiutyk <trofimich@gmail.com>
SPDX-License-Identifier: MIT
License: https://opensource.org/license/mit
*)

(*!
<summary>Serializes configuration objects into a JSON document.</summary>
<description>
The instance owns its native SAX writer. Use sequentially from one task without reentry.
WriteValue validates the source address, type and size before emitting a field. WSTRING values produce JSON text.
The writer does not track key uniqueness or nesting depth; maintaining unique property names and balanced
object/array calls is the responsibility of the caller. Structural violations are propagated from the native writer.
</description>
*)

{attribute 'no_explicit_call' := 'do not call this function block directly'}
FUNCTION_BLOCK JsonConfigurationWriter EXTENDS TOF_Core.Object IMPLEMENTS TOF_Core.IConfigurationWriter
VAR CONSTANT
	// Standard HRESULT for an invalid writer operand.
	_InvalidArgument : HRESULT := TO_DINT(16#80070057);
	// Standard HRESULT for a failed operation without a native error code.
	_UnspecifiedFailure : HRESULT := TO_DINT(16#80004005);
END_VAR
VAR_STAT
	_ClassName : STRING := __POUNAME();
END_VAR
VAR
	_Writer : Tc3_JsonXml.FB_JsonSaxWriter;
	_Converter : Tc3_JsonXml.FB_JsonReadWriteDatatype;
	_Utf8Value : TOF_Core.JSON_DOCUMENT;
END_VAR

(*!
<summary>Opens an ordered list.</summary>
<description>
Writes a property key when name is nonempty, then opens a JSON array. Property names within an enclosing object
must be unique. Propagates native writer errors to the active serialization call.
</description>
<param name="name">List property name, or empty for array items or root.</param>
*)
METHOD BeginArray
VAR_INPUT
	name : STRING;
END_VAR
IF name <> '' THEN
	// Tc3_JsonXml.FB_JsonSaxWriter.AddKey returns VOID; state errors are caught by subsequent calls.
	_Writer.AddKey(key := name);
END_IF

checkResult(result := _Writer.StartArray());
END_METHOD

(*!
<summary>Resets the native writer and opens the document root object.</summary>
<description>Prepares writer for streaming a fresh configuration object.</description>
*)
METHOD BeginDocument
checkResult(result := _Writer.ResetDocument());
BeginObject(name := '');
END_METHOD

(*!
<summary>Opens an object.</summary>
<description>
Writes a property key when name is nonempty, then opens a JSON object. Property names within an enclosing object
must be unique. Propagates native writer errors to the active serialization call.
</description>
<param name="name">Object property name, or empty for array items or root.</param>
*)
METHOD BeginObject
VAR_INPUT
	name : STRING;
END_VAR
IF name <> '' THEN
	// Tc3_JsonXml.FB_JsonSaxWriter.AddKey returns VOID; state errors are caught by subsequent calls.
	_Writer.AddKey(key := name);
END_IF

checkResult(result := _Writer.StartObject());
END_METHOD

(*!
<summary>Propagates a native writer failure.</summary>
<description>
A nonzero result raises StandardException with the original HRESULT. For value conversion failures the
diagnostic includes the field name and native datatype. The caller discards an incomplete document.
</description>
<param name="result">HRESULT returned by the native writer operation.</param>
<param name="name">Value property name, or empty for array items.</param>
<param name="typeName">Native datatype name for value conversion, or empty for other operations.</param>
*)
METHOD PRIVATE checkResult
VAR_INPUT
	result : HRESULT;
	name : STRING := '';
	typeName : STRING := '';
END_VAR
VAR
	message : TOF_Core.ERROR_MESSAGE;
END_VAR
IF result = 0 THEN
	RETURN;
END_IF

message := "Cannot write configuration document";

IF typeName <> '' THEN
	message := TOF_Core.WideStrings.Concat255(
		"Cannot write configuration value '",
		TO_WSTRING(name),
		"' using native datatype '",
		TO_WSTRING(typeName),
		"'"
	);
END_IF

TOF_Core.Exceptions.ThrowStandard(
	sourceNamespaceName := NamespaceName,
	sourceClassName := ClassName,
	sourcePOUName := __POUNAME(),
	sourcePosition := __POSITION(),
	message := message,
	errorCode := TO_UDINT(result)
);
END_METHOD

(*!
<summary>Provides the concrete serializer class name.</summary>
<description>Borrows read-only instance storage that remains valid for the instance lifetime.</description>
*)
{attribute 'monitoring' := 'call'}
PROPERTY ClassName : REFERENCE TO STRING
GET
ClassName REF= _ClassName;
END_GET
END_PROPERTY

(*!
<summary>Closes the current list.</summary>
<description>Propagates native writer errors to the active serialization call.</description>
*)
METHOD EndArray
checkResult(result := _Writer.EndArray());
END_METHOD

(*!
<summary>Closes the root object and extracts the serialized JSON document text.</summary>
<description>Copies output text into document. An incomplete or zero-length result raises.</description>
<param name="document">Destination text buffer for the JSON document.</param>
*)
METHOD EndDocument
VAR_IN_OUT
	document : TOF_Core.JSON_DOCUMENT;
END_VAR
VAR
	result : HRESULT;
	length : UDINT;
END_VAR
EndObject();
length := _Writer.CopyDocument(pDoc := document, nDoc := SIZEOF(document), hrErrorCode => result);
checkResult(result := result);

IF length = 0 THEN
	checkResult(result := _UnspecifiedFailure);
END_IF
END_METHOD

(*!
<summary>Closes the current object.</summary>
<description>Propagates native writer errors to the active serialization call.</description>
*)
METHOD EndObject
checkResult(result := _Writer.EndObject());
END_METHOD

(*!
<summary>Provides the compiler-initialized library namespace.</summary>
<description>Borrows read-only library storage; no allocation or ownership transfer occurs.</description>
*)
{attribute 'monitoring' := 'call'}
PROPERTY NamespaceName : REFERENCE TO STRING
GET
NamespaceName REF= CurrentNamespace.Name;
END_GET
END_PROPERTY

(*!
<summary>Reports the complete instance size in bytes.</summary>
<description>Uses XSIZEOF; separately allocated native resources are not included.</description>
*)
{attribute 'monitoring' := 'call'}
PROPERTY SelfSize : ULINT
GET
SelfSize := XSIZEOF(THIS^);
END_GET
END_PROPERTY

(*!
<summary>Writes a fresh JSON document from a serializable configuration object.</summary>
<description>
Accepts any object implementing IConfigurationSerializable. Use from one task without reentry. Only consume
the destination after normal return; on failure document is cleared before writing and must be discarded.
Each call resets the native writer before invoking source.Serialize.
</description>
<param name="source">Configuration source to serialize.</param>
<param name="document">Destination text buffer for the JSON document.</param>
*)
METHOD Serialize
VAR_INPUT
	source : TOF_Core.IConfigurationSerializable;
END_VAR
VAR_IN_OUT
	document : TOF_Core.JSON_DOCUMENT;
END_VAR
document := '';

IF source = 0 THEN
	checkResult(result := _InvalidArgument);
END_IF

BeginDocument();
source.Serialize(writer := THIS^);
EndDocument(document := document);
END_METHOD

(*!
<summary>Copies one elementary IEC value.</summary>
<description>
Rejects a null source or invalid type/size before writing a key. These validation failures preserve the document.
For WSTRING, converts the text up to its first null word to UTF-8 before writing the optional key.
An unterminated source or incomplete conversion raises StandardException.
Writes the value after its optional key. Property names within an enclosing
object must be unique. Propagates native writer errors to the active serialization call. A native value conversion
failure reports the field name and requested native datatype.
</description>
<param name="name">Value property name, or empty for array items.</param>
<param name="valueType">Elementary IEC type class.</param>
<param name="data">Pointer to readable source memory.</param>
<param name="size">Source memory size in bytes.</param>
*)
METHOD WriteValue
VAR_INPUT
	name : STRING;
	valueType : TOF_Core.CONFIGURATION_VALUE_TYPE;
	data : PVOID;
	size : UDINT;
END_VAR
VAR
	typeName : STRING;
	written : BOOL;
	sourceWords : POINTER TO WORD;
	wordCount : UDINT;
	textLength : UDINT;
	result : HRESULT;
END_VAR
IF data = 0 OR_ELSE size = 0 THEN
	checkResult(result := _InvalidArgument);
END_IF

typeName := JsonDatatypes.ToDatatypeName(valueType := valueType, size := size);

IF typeName = '' THEN
	checkResult(result := _InvalidArgument);
END_IF

IF valueType = TOF_Core.CONFIGURATION_VALUE_TYPE.TYPE_WSTRING THEN
	sourceWords := data;
	wordCount := size / TOF_Core.WideStrings.CharSize;

	WHILE textLength < wordCount AND_THEN sourceWords[textLength] <> 0 DO
		textLength := textLength + 1;
	END_WHILE

	IF textLength = wordCount THEN
		checkResult(result := _InvalidArgument, name := name, typeName := typeName);
	END_IF

	_Utf8Value := '';

	IF textLength > 0 THEN
		IF NOT Tc2_Utilities.WSTRING_TO_UTF8(
			pDstUTF8 := ADR(_Utf8Value),
			pSrcWSTRING := data,
			nDstSize := SIZEOF(_Utf8Value)
		) OR_ELSE Tc2_Utilities.UTF8Len(pUTF8 := ADR(_Utf8Value)) <> textLength
		THEN
			checkResult(result := _InvalidArgument, name := name, typeName := typeName);
		END_IF
	END_IF
END_IF

IF name <> '' THEN
	// Tc3_JsonXml.FB_JsonSaxWriter.AddKey returns VOID; state errors are caught by subsequent calls.
	_Writer.AddKey(key := name);
END_IF

IF valueType = TOF_Core.CONFIGURATION_VALUE_TYPE.TYPE_WSTRING THEN
	_Writer.AddString(value := _Utf8Value);
	RETURN;
END_IF

written := _Converter.AddJsonValueFromSymbol(
	fbWriter := _Writer,
	sDatatype := typeName,
	nData := size,
	pData := data,
	hrErrorCode => result
);

IF NOT written AND_THEN result = 0 THEN
	result := _UnspecifiedFailure;
END_IF

checkResult(result := result, name := name, typeName := typeName);
END_METHOD

END_FUNCTION_BLOCK
